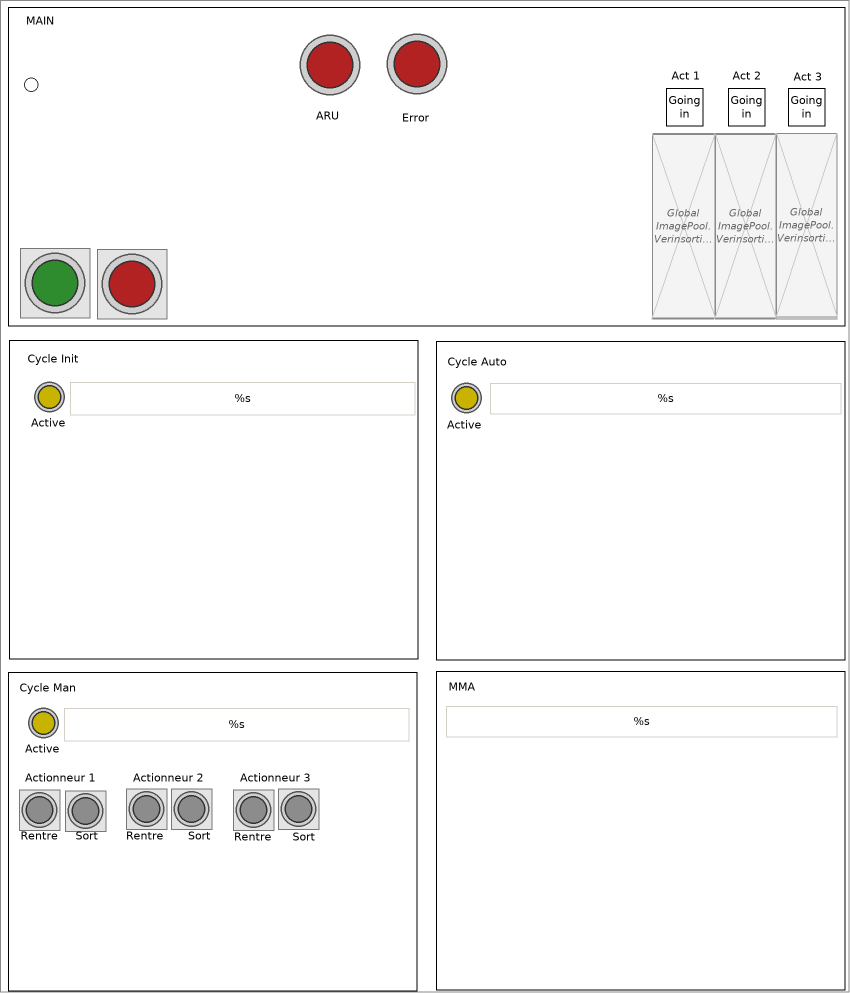
VISUALIZATION Visualization  // 850x993
    Rectangle (9,340 409x319)
    Lamp1 (31,379 37x36), variable: fbCycleInit.xBusy, style: Lamp-Lamp1-Yellow
    Label (13,344 80x30), "Cycle Init"
    Label (19,408 59x30), "Active"
    Rectangle (436,341 409x319)
    Label (437,347 80x30), "Cycle Auto"
    Lamp1 (448,380 37x36), variable: fbCycleAuto.xBusy, style: Lamp-Lamp1-Yellow
    Label (435,410 59x30), "Active"
    Textfield (490,383 351x31), "%s", text variable: fbCycleAuto.fbEtape.sMess
    Textfield (70,382 345x33), "%s", text variable: MAIN.fbCycleInit.fbEtape.sMess
    Rectangle (8,7 837x319)
    Label (0,6 80x30), "MAIN"
    Rectangle (8,672 409x319)
    Rectangle (436,671 409x319)
    Label (8,673 80x30), "Cycle Man"
    Label (422,672 80x30), "MMA"
    Textfield (446,706 391x31), "%s", text variable: fbMMA.fbEtape.sMess
    Label (13,734 59x30), "Active"
    Lamp1 (25,705 37x36), variable: fbCycleMan.xBusy, style: Lamp-Lamp1-Yellow
    Textfield (64,708 345x33), "%s", text variable: MAIN.fbCycleMan.fbEtape.sMess
    Lamp1 (382,29 70x70), variable: stParam.stStatus.xErreur, style: Lamp-Lamp1-Red
    Label (386,103 59x30), "Error"
    Lamp1 (295,30 70x70), variable: fbBtn.xAru=0, style: Lamp-Lamp1-Red
    Label (298,101 59x30), "ARU"
    PushSwitch (19,788 41x44), variable: fbBtn.xManAct1Rentre, behaviour: TAP, style: Switch-PushSwitch-Gray
    PushSwitch (65,789 41x44), variable: fbBtn.xManAct1Sort, behaviour: TAP, style: Switch-PushSwitch-Gray
    Label (4,821 111x30), "Rentre Sort"
    PushSwitch (171,787 41x44), variable: fbBtn.xManAct2Sort, behaviour: TAP, style: Switch-PushSwitch-Gray
    PushSwitch (126,787 41x44), variable: fbBtn.xManAct2Rentre, behaviour: TAP, style: Switch-PushSwitch-Gray
    Label (113,821 111x30), "Rentre Sort"
    PushSwitch (278,787 41x44), variable: fbBtn.xManAct3Sort, behaviour: TAP, style: Switch-PushSwitch-Gray
    PushSwitch (233,788 41x44), variable: fbBtn.xManAct3Rentre, behaviour: TAP, style: Switch-PushSwitch-Gray
    Label (219,822 111x30), "Rentre Sort"
    RadioButton (22,36 150x97), variable: stParam.stStatus.eMMA
        Areas[0]: Text=Mode Init
        Areas[1]: Text=Mode Auto
        Areas[2]: Text=Mode Manual
    Label (5,763 111x30), "Actionneur 1"
    Label (113,763 111x30), "Actionneur 2"
    Label (220,763 111x30), "Actionneur 3"
    Label (646,61 80x30), "Act 1"
    Label (707,61 80x30), "Act 2"
    Label (768,62 80x30), "Act 3"
    Image (775,133 62x186), invisible if: fbAct3.xInInPos=0, image: GlobalImagePool.Verinrentree2
    Image (713,133 62x186), invisible if: fbAct2.xInInPos=0, image: GlobalImagePool.Verinrentree2
    Image (652,133 62x186), invisible if: fbAct1.xInInPos=0, image: GlobalImagePool.Verinrentree2
    Image (652,134 63x184), invisible if: fbAct1.xInOutPos=0, image: GlobalImagePool.Verinsortie2
    Image (715,134 61x184), invisible if: fbAct2.xInOutPos=0, image: GlobalImagePool.Verinsortie2
    Image (776,133 61x184), invisible if: fbAct3.xInOutPos=0, image: GlobalImagePool.Verinsortie2
    Rectangle (788,88 37x38), "Going out", invisible if: fbAct3.xGoingOutNow=0
    Rectangle (728,88 37x38), "Going out", invisible if: fbAct2.xGoingOutNow=0
    Rectangle (666,88 37x38), "Going out", invisible if: fbAct1.xGoingOutNow=0
    Rectangle (666,88 37x38), "Going in", invisible if: fbAct1.xGoingInNow=0
    Rectangle (788,88 37x38), "Going in", invisible if: fbAct3.xGoingInNow=0
    Rectangle (728,88 37x38), "Going in", invisible if: fbAct2.xGoingInNow=0
    PushSwitch (20,248 70x70), tooltip "Start", variable: fbBtn.xStart, behaviour: TAP, style: Switch-PushSwitch-Green
    PushSwitch (97,249 70x70), tooltip "Stop", variable: fbBtn.xStop, invisible if: fbMMA.iEtape<>350, behaviour: TAP, style: Switch-PushSwitch-Red
END_VISUALIZATION

(* stored: Version 1.1.0.1, ProductVersion 3.1.4020.6
   Visu Visualization: Id {1e4c2f99-d035-41f9-adba-3d4322eca24e} *)
